      val_new := Roots.PolyEval(ADR(polynom), 5, tz);
      IF (ABS(val_new) < 64 * ABS(Roots.PolyEval(ADR(dderiv), 3, tz)) * Constants.Tolerance)
      THEN
        root[rootCount+1] := tz;
        rootCount := rootCount + 1;
      ELSIF (Roots.PolyEval(ADR(polynom), 5, tz_current) * val_new < 0)
      THEN
        root[rootCount+1] := Roots.ShrinkInterval(ADR(polynom), 5, tz_current, tz);
        rootCount := rootCount + 1;
      END_IF
    
      tz_current := tz;
    END_FOR
  
    val_max := Roots.PolyEval(ADR(polynom), 5, tz_max);
    IF Roots.PolyEval(ADR(polynom), 5, tz_current) * val_max < 0
    THEN
      root[rootCount+1] := Roots.ShrinkInterval(ADR(polynom), 5, tz_current, tz_max);
      rootCount := rootCount + 1;
    ELSIF ABS(val_max) < 8 * Constants.DoubleEpsilon
    THEN
      root[rootCount+1] := tz_max;
      rootCount := rootCount + 1;
    END_IF

    FOR i:=0 TO rootCount
    DO
      t := root[i];
      IF t < 0.0
      THEN
        CONTINUE;
      END_IF
    
      h1 := (a0_a0 + af_af)*0.5 + jMax*(2*a0*t + jMax*t*t - vd);
      IF h1 < 0
      THEN
        CONTINUE;
      END_IF
    
      IF ABS(jMax) < Constants.DoubleEpsilon
      THEN
        CONTINUE;
  		END_IF
    
      h1 := SQRT(h1)/ABS(jMax);
      orig := -pd - (2*a0_p3 + 4*af_p3 + 24*a0*jMax*t*(af + jMax*(h1 + t - tf)) + 6*a0_a0*(af + jMax*(2*t - tf)) + 6*(a0_a0 + af_af)*jMax*h1 + 12*af*jMax*(jMax*t*t - vd) + 12*jMax_jMax*(jMax*t*t*(h1 + t - tf) - tf*v0 - h1*vd))/(12*jMax_jMax);
      deriv_newton := -(a0 + jMax*t)*(3*(h1 + t) - 2*tf + (a0 + 2*af)/jMax);
    
      IF orig <> orig OR_ELSE deriv_newton <> deriv_newton OR_ELSE ABS(deriv_newton) < Constants.DoubleEpsilon 
      THEN
        CONTINUE;
      END_IF
    
      t := t - orig / deriv_newton;
  
      IF t > tf OR_ELSE t <> t (*isnan*)
      THEN
        CONTINUE;
      END_IF
  
      h1 := (a0_a0 + af_af)/(2*jMax_jMax) + (t*(2*a0 + jMax*t) - vd)/jMax;
      IF h1 >= 0
      THEN
        h1 := SQRT(h1);
    
        Profile.t[0] := t;
        Profile.t[1] := 0;
        Profile.t[2] := t + a0/jMax;
        Profile.t[3] := tf - 2*(t + h1) - (a0 + af)/jMax;
        Profile.t[4] := h1;
        Profile.t[5] := 0;
        Profile.t[6] := h1 + af/jMax;
    
        time_vel := Profile.CheckWithTiming(ProfileControlSigns.Uddu, ReachedLimits.vel, tf, jMax, vMax, vMin, aMax, aMin);
        IF time_vel
        THEN
          RETURN;
        END_IF
      END_IF
    END_FOR
  END_IF
  
  // Profile UDUD
  ph1 := af_af - 2*jMax*(2*af*tf + jMax*tf_tf - 3*vd);
  ph2 := af_p3 - 3*jMax_jMax*g1 + 3*af*jMax*vd;
  ph3 := 2*jMax*tf*g1 + 3*vd_vd;
  ph4 := af_p4 - 8*af_p3*jMax*tf + 12*jMax*(jMax*ph3 + af_af*vd + 2*af*jMax*(g1 - tf*vd));
  ph5 := af + jMax*tf;
  
  // Find root of 6th order polynom
  polynom[0] := 1.0;
  polynom[1] := (5*a0 - ph5)/jMax;
  polynom[2] := (39*a0_a0 - ph1 - 16*a0*ph5)/(4*jMax_jMax);
  polynom[3] := (55*a0_p3 - 33*a0_a0*ph5 - 6*a0*ph1 + 2*ph2)/(6*jMax_jMax*jMax);
  polynom[4] := (101*a0_p4 + ph4 - 76*a0_p3*ph5 - 30*a0_a0*ph1 + 16*a0*ph2)/(24*jMax_jMax*jMax_jMax);
  polynom[5] := (a0*(11*a0_p4 + ph4 - 10*a0_p3*ph5 - 6*a0_a0*ph1 + 4*a0*ph2))/(12*jMax_jMax*jMax_jMax*jMax);
  polynom[6] := (11*a0_p6 - af_p6 - 12*a0_p5*ph5 - 48*af_p3*jMax_jMax*g1 - 9*a0_p4*ph1 + 72*jMax_jMax*jMax*(jMax*g1*g1 - vd_vd*vd - 2*af*g1*vd) - 6*af_p4*jMax*vd - 36*af_af*jMax_jMax*vd_vd + 8*a0_p3*ph2 + 3*a0_a0*ph4)/(144*jMax_jMax*jMax_jMax*jMax_jMax);
  
  Roots.PolyMonicDeri(ADR(polynom), 6, out:=ADR(deriva));
  Roots.PolyMonicDeri(ADR(deriva), 5, out:=ADR(dderiv));
  Roots.SolveQuartMonic(ADR(dderiv[1]), 4, rootCount:=rootCount, roots:=root);
  
  tz_min := 0.0;
  tz_max := tf;
  dd_tz_current := tz_min;
  
  FOR i:=0 TO rootCount
  DO
    tz := root[i];
    IF tz >= tz_max
    THEN
      CONTINUE;
    END_IF
    
    orig := Roots.PolyEval(ADR(dderiv), 4, tz);
    IF (ABS(orig) > Constants.Tolerance)
    THEN
      Roots.PolyMonicDeri(ADR(dderiv), 4, out:=ADR(ddderiv));   
      res := Roots.PolyEval(ADR(ddderiv), 3, tz);
      IF ABS(res) > Constants.DoubleEpsilon
      THEN
        tz := tz - orig / res;
      END_IF
    END_IF  
  
    IF (Roots.PolyEval(ADR(deriva), 5, dd_tz_current) * Roots.PolyEval(ADR(deriva), 5, tz) < 0)
    THEN
      dd_tz_intervals[dd_tz_intervalCount+1, 0] := dd_tz_current;
      dd_tz_intervals[dd_tz_intervalCount+1, 1] := tz;
      dd_tz_intervalCount := dd_tz_intervalCount + 1;
    END_IF
  
    dd_tz_current := tz;
      
  END_FOR
  
  IF (Roots.PolyEval(ADR(deriva), 5, dd_tz_current) * Roots.PolyEval(ADR(deriva), 5, tz_max) < 0)
  THEN
    dd_tz_intervals[dd_tz_intervalCount+1, 0] := dd_tz_current; 
    dd_tz_intervals[dd_tz_intervalCount+1, 1] := tz_max;
    dd_tz_intervalCount := dd_tz_intervalCount + 1;
  END_IF
  
  rootCount := -1;
  tz_current := tz_min;
  FOR i:=0 TO dd_tz_intervalCount
  DO
    tz := Roots.ShrinkInterval(ADR(deriva), 5, dd_tz_intervals[i, 0], dd_tz_intervals[i, 1]);
    IF tz >= tz_max
    THEN
      CONTINUE;
    END_IF
    
    p_val := Roots.PolyEval(ADR(polynom), 6, tz);
    IF (ABS(p_val) < 64 * ABS(Roots.PolyEval(ADR(dderiv), 4, tz)) * Constants.Tolerance)
    THEN
      root[rootCount+1] := tz;
      rootCount := rootCount + 1;
    ELSIF (Roots.PolyEval(ADR(polynom), 6, tz_current) * p_val < 0)
    THEN
      root[rootCount+1] := Roots.ShrinkInterval(ADR(polynom), 6, tz_current, tz);
      rootCount := rootCount + 1;
    END_IF
    tz_current := tz;
  END_FOR
  
  IF (Roots.PolyEval(ADR(polynom), 6, tz_current) * Roots.PolyEval(ADR(polynom), 6, tz_max) < 0)
  THEN
    root[rootCount+1] := Roots.ShrinkInterval(ADR(polynom), 6, tz_current, tz_max);
    rootCount := rootCount + 1;
  END_IF
  
  
  FOR i:=0 TO rootCount
  DO
    t := root[i];
    
    // Double Newton step (regarding pd)
    h1 := (af_af - a0_a0)/(2*jMax_jMax) - ((2*a0 + jMax*t)*t - vd)/jMax;
    IF h1 < 0
    THEN
      CONTINUE;
    END_IF
    
    h1 := SQRT(h1);
    orig := -pd + (af_p3 - a0_p3 + 3*a0_a0*jMax*(tf - 2*t))/(6*jMax_jMax) + (2*a0 + jMax*t)*t*(tf - t) + (jMax*h1 - af)*h1*h1 + tf*v0;
    deriv_newton := (a0 + jMax*t)*(2*(af + jMax*tf) - 3*jMax*(h1 + t) - a0)/jMax;
  
    IF ABS(deriv_newton) <= Constants.DoubleEpsilon
    THEN
      CONTINUE;
    END_IF
    
    t := t - orig / deriv_newton;
    h1 := (af_af - a0_a0)*0.5 - jMax*((2*a0 + jMax*t)*t - vd);
    IF h1 < 0
    THEN
      CONTINUE;
    END_IF
    h1 := SQRT(h1)/ABS(jMax);  
    orig := -pd + (af_p3 - a0_p3 + 3*a0_a0*jMax*(tf - 2*t))/(6*jMax_jMax) + (2*a0 + jMax*t)*t*(tf - t) + (jMax*h1 - af)*h1*h1 + tf*v0;
    IF (ABS(orig) > 1E-9)
    THEN
      deriv_newton := (a0 + jMax*t)*(2*(af + jMax*tf) - 3*jMax*(h1 + t) - a0)/jMax;
      
      IF ABS(deriv_newton) <= Constants.DoubleEpsilon
      THEN
        CONTINUE;
      END_IF
      
      t := t - orig / deriv_newton;           
    END_IF
  
    h1 := (af_af - a0_a0)*0.5 - jMax*((2*a0 + jMax*t)*t - vd);
    IF h1 < 0
    THEN
      CONTINUE;
    END_IF
    h1 := SQRT(h1)/ABS(jMax);
    Profile.t[0] := t;
    Profile.t[1] := 0;
    Profile.t[2] := t + a0/jMax;
    Profile.t[3] := tf - 2*(t + h1) + ad/jMax;
    Profile.t[4] := h1;
    Profile.t[5] := 0;
    Profile.t[6] := h1 - af/jMax;
  
    time_vel := Profile.CheckWithTiming(ProfileControlSigns.Udud, ReachedLimits.Vel, tf, jMax, vMax, vMin, aMax, aMin);
    IF time_vel
    THEN
      RETURN;
    END_IF
  END_FOR
END_IF
END_METHOD

END_FUNCTION_BLOCK

// ---- Struckig/Math/Power2.TcPOU
// Struckig
// Copyright (C) 2022 Stefan Besler

// This program is free software: you can redistribute it and/or modify
// it under the terms of the GNU General Public License as published by
// the Free Software Foundation, either version 3 of the License, or
// (at your option) any later version.

// This program is distributed in the hope that it will be useful,
// but WITHOUT ANY WARRANTY; without even the implied warranty of
// MERCHANTABILITY or FITNESS FOR A PARTICULAR PURPOSE.  See the
// GNU General Public License for more details.
//
// You should have received a copy of the GNU General Public License
// along with THIS PROGRAM.  IF NOT, see <http://www.gnu.org/licenses/>.
/// Internal square helper.
/// Returns `v * v`.
FUNCTION INTERNAL Power2 : LREAL
VAR_INPUT
  v : LREAL; //< Input value.
END_VAR

Power2 := v*v;

END_FUNCTION

// ---- Struckig/Velocity/VelocityThirdOrderStep1.TcPOU
// Struckig
// Copyright (C) 2022 Stefan Besler

// This program is free software: you can redistribute it and/or modify
// it under the terms of the GNU General Public License as published by
// the Free Software Foundation, either version 3 of the License, or
// (at your option) any later version.

// This program is distributed in the hope that it will be useful,
// but WITHOUT ANY WARRANTY; without even the implied warranty of
// MERCHANTABILITY or FITNESS FOR A PARTICULAR PURPOSE.  See the
// GNU General Public License for more details.
//
// You should have received a copy of the GNU General Public License
// along with THIS PROGRAM.  IF NOT, see <http://www.gnu.org/licenses/>.
/// Mathematical equations for Step 1 in third-order velocity interface: Extremal profiles
FUNCTION_BLOCK INTERNAL VelocityThirdOrderStep1 
VAR
  a0, af : LREAL;
  aMax, aMin, jMax : LREAL;
  vd : LREAL;
  
  ValidProfiles : ARRAY[0..2] OF ProfileDesc; // Max 3 valid profiles
  ValidProfileCount : INT := -1;  
END_VAR

METHOD AddInterval
VAR_INPUT
  interval : REFERENCE TO BlockInterval;
  Left : REFERENCE TO ProfileDesc;
  Right : REFERENCE TO ProfileDesc;
END_VAR
VAR_INST
  left_duration,right_duration : LREAL;   
END_VAR
left_duration := Left.t_sum[6] + Left.Brake.Duration + Left.Accel.Duration; 
right_duration := Right.t_sum[6] + Right.Brake.Duration + Right.Accel.Duration; 
IF (left_duration < right_duration)
THEN
  interval.Left := left_duration;
  interval.Right := right_duration;
  interval.Profile := Right;
  interval.IsUsed := TRUE;
ELSE
  interval.Left := right_duration;
  interval.Right := left_duration;
  interval.Profile := Left;
  interval.IsUsed := TRUE;
END_IF
END_METHOD

METHOD AddProfile
VAR_IN_OUT CONSTANT
  Profile : ProfileDesc;
END_VAR
ValidProfileCount := ValidProfileCount + 1;
ValidProfiles[ValidProfileCount] := Profile;
ValidProfiles[ValidProfileCount].pf := Profile.p[7];
END_METHOD

METHOD CalculateBlock : BOOL
VAR_INPUT
  block : REFERENCE TO Block;
END_VAR
VAR
  i, j : INT;
  Tmin : LREAL;
  idx_min : INT;
  idx_else_1, idx_else_2, idx_else_3, idx_else_4 : INT;
END_VAR
IF (ValidProfileCount = 0) OR_ELSE (ValidProfileCount = 1 AND_THEN ABS(ValidProfiles[0].t_sum[6] - ValidProfiles[1].t_sum[6]) < 8*Constants.Epsilon)
THEN
  block.Pmin := ValidProfiles[0];
  block.Tmin := block.Pmin.t_sum[6] + block.Pmin.Brake.Duration + block.Pmin.Accel.Duration;  
  CalculateBlock := TRUE;
  RETURN;
// Only happens due to numerical issues
ELSIF (ValidProfileCount = 3) 
THEN
  // Find "identical" profiles
  IF (ABS(ValidProfiles[0].t_sum[6] - ValidProfiles[1].t_sum[6]) < 16*Constants.Epsilon OR_ELSE ValidProfiles[0].Direction <> ValidProfiles[1].Direction)
  THEN
    RemoveProfile(1);
  ELSIF (ABS(ValidProfiles[1].t_sum[6] - ValidProfiles[2].t_sum[6]) < 16*Constants.Epsilon  OR_ELSE ValidProfiles[2].Direction <> ValidProfiles[2].Direction)
  THEN
    RemoveProfile(2);
  ELSIF (ABS(ValidProfiles[0].t_sum[6] - ValidProfiles[2].t_sum[6]) < 256*Constants.Epsilon OR_ELSE ValidProfiles[0].Direction <> ValidProfiles[2].Direction)
  THEN
    RemoveProfile(2);
  ELSE
    RETURN;
  END_IF

ELSIF ((ValidProfileCount+1) MOD 2 = 0)
THEN
  RETURN;
END_IF

// Find index of fastest Profile
Tmin := Constants.Infinity;
FOR i:=0 TO ValidProfileCount
DO
  FOR j:=0 TO ValidProfileCount
  DO
    IF ValidProfiles[i].t_sum[6] + ValidProfiles[i].Brake.Duration < ValidProfiles[j].t_sum[6] + ValidProfiles[j].Brake.Duration AND_THEN
       ValidProfiles[i].t_sum[6] + ValidProfiles[i].Brake.Duration < Tmin
    THEN
      Tmin := ValidProfiles[i].t_sum[6] + ValidProfiles[i].Brake.Duration + ValidProfiles[i].Accel.Duration;
      idx_min := i;
		END_IF
  END_FOR
END_FOR

block.Pmin := ValidProfiles[idx_min];
block.Tmin := block.Pmin.t_sum[6] + block.Pmin.Brake.Duration + block.Pmin.Accel.Duration;  

IF (ValidProfileCount = 2)
THEN
  idx_else_1 := (idx_min + 1) MOD 3;
  idx_else_2 := (idx_min + 2) MOD 3;
  
  AddInterval(block.A, ValidProfiles[idx_else_1], ValidProfiles[idx_else_2]);
  CalculateBlock := TRUE;
  RETURN;

 ELSIF (ValidProfileCount = 4)
 THEN
  idx_else_1 := (idx_min + 1) MOD 5;
  idx_else_2 := (idx_min + 2) MOD 5;
  idx_else_3 := (idx_min + 3) MOD 5;
  idx_else_4 := (idx_min + 4) MOD 5;
  
  IF (ValidProfiles[idx_else_1].Direction = ValidProfiles[idx_else_2].Direction)
  THEN
    AddInterval(block.A, ValidProfiles[idx_else_1], ValidProfiles[idx_else_2]);
    AddInterval(block.B, ValidProfiles[idx_else_3], ValidProfiles[idx_else_4]);
  ELSE 
    AddInterval(block.A, ValidProfiles[idx_else_1], ValidProfiles[idx_else_4]);
    AddInterval(block.B, ValidProfiles[idx_else_2], ValidProfiles[idx_else_3]);
  END_IF
  
  CalculateBlock := TRUE;
  RETURN;
END_IF
END_METHOD

METHOD Get : BOOL
VAR_INPUT
  input : ProfileDesc;
END_VAR
VAR_IN_OUT
  block : Block; 
END_VAR
VAR
  aMax, aMin, jMax : LREAL;
END_VAR
ValidProfileCount := -1;

// Zero-limits special case
IF THIS^.jMax = 0.0
THEN
  block.Pmin.SetBoundary(input);
  
  IF time_all_single_step(block.Pmin, THIS^.aMax, THIS^.aMin, THIS^.jMax)
  THEN
    block.Tmin := block.Pmin.t_sum[6] + block.Pmin.Brake.Duration + block.Pmin.Accel.Duration;
    AddInterval(block.A, block.Pmin, block.Pmin);
    IF ABS(a0) > Constants.DoubleEpsilon
    THEN
	  block.A.Left := block.Tmin;
      block.A.Right := Constants.Infinity;
    END_IF
    
    Get := TRUE;
    RETURN; 
	END_IF
  
  RETURN;  
END_IF

validProfiles[0].SetBoundary(input);

IF ABS(af) < Constants.DoubleEpsilon
THEN
  // There is no blocked interval when af==0, so return after first found profile
  aMax := SEL((vd >= 0), THIS^.aMin, THIS^.aMax);
  aMin := SEL((vd >= 0), THIS^.aMax, THIS^.aMin);
  jMax := SEL((vd >= 0), -THIS^.jMax, THIS^.jMax);
  
  time_none(input, aMax, aMin, jMax, TRUE);
  IF ValidProfileCount >= 0
  THEN 
    Get := CalculateBlock(block);
    RETURN;
	END_IF
  
  time_acc0(input, aMax, aMin, jMax, TRUE);
  IF ValidProfileCount >= 0
  THEN 
    Get := CalculateBlock(block);
    RETURN;
	END_IF
  
  time_none(input, aMin, aMax, -jMax, TRUE);
  IF ValidProfileCount >= 0
  THEN 
    Get := CalculateBlock(block);
    RETURN;
	END_IF
  
  time_acc0(input, aMin, aMax, -jMax, TRUE);
ELSE
  time_none(input, THIS^.aMax, THIS^.aMin, THIS^.jMax, FALSE);
  time_none(input, THIS^.aMin, THIS^.aMax, -THIS^.jMax, FALSE);
  time_acc0(input, THIS^.aMax, THIS^.aMin, THIS^.jMax, FALSE);
  time_acc0(input, THIS^.aMin, THIS^.aMax, -THIS^.jMax, FALSE);
END_IF

Get := CalculateBlock(block);
END_METHOD

METHOD PRIVATE RemoveProfile : BOOL
VAR_INPUT
  index : INT;
END_VAR
VAR
  i : INT;
END_VAR
// todo, this is pretty slow in twincat
FOR i:=index TO ValidProfileCount-2
DO
  ValidProfiles[i] := ValidProfiles[i + 1];
END_FOR

ValidProfileCount := ValidProfileCount - 1;
END_METHOD

METHOD Set
VAR_INPUT
  v0, a0 : LREAL; 
  vf, af : LREAL; 
  aMax, aMin : LREAL; 
  jMax : LREAL;   
END_VAR
THIS^.a0 := a0;
THIS^.vd := vf - v0;
THIS^.af := af;;
THIS^.aMax := aMax;
THIS^.aMin := aMin;
THIS^.jMax := jMax;
END_METHOD

METHOD PRIVATE time_acc0
VAR_IN_OUT
  profile : ProfileDesc;
END_VAR
VAR_INPUT
  aMax, aMin, jMax : LREAL;
  return_after_found : BOOL;  
END_VAR
// UD
profile.t[0] := (-a0 + aMax)/jMax;
profile.t[1] := (a0*a0 + af*af - 2*aMax*aMax + 2*jMax*vd)/(2*aMax*jMax);
profile.t[2] := (-af + aMax)/jMax;
profile.t[3] := 0;
profile.t[4] := 0;
profile.t[5] := 0;
profile.t[6] := 0;

IF (Profile.CheckForVelocity(ProfileControlSigns.Uddu, ReachedLimits.Acc0, jMax, aMax, aMin))
THEN
  AddProfile(profile);
  IF return_after_found
  THEN
    RETURN;
	END_IF
END_IF
END_METHOD

METHOD PRIVATE time_all_single_step : BOOL
VAR_IN_OUT
  profile : ProfileDesc;
END_VAR
VAR_INPUT
  aMax, aMin, jMax : LREAL;
END_VAR
IF ABS(af - a0) > Constants.DoubleEpsilon
THEN 
  RETURN;
END_IF
    
profile.t[0] := 0;
profile.t[1] := 0;
profile.t[2] := 0;
profile.t[3] := 0;
profile.t[4] := 0;
profile.t[5] := 0;
profile.t[6] := 0;

IF ABS(a0) > Constants.DoubleEpsilon
THEN

  IF ABS(a0) > Constants.DoubleEpsilon
  THEN
    profile.t[3] := vd / a0;
    IF profile.CheckForVelocity(ProfileControlSigns.uddu, ReachedLimits.None, 0.0, aMax, aMin)
    THEN
      time_all_single_step := TRUE;
      RETURN;
    END_IF
	END_IF

 ELSE IF ABS(vd) < Constants.DoubleEpsilon
 THEN
    IF profile.CheckForVelocity(ProfileControlSigns.uddu, ReachedLimits.None, 0.0, aMax, aMin)
    THEN 
      time_all_single_step := TRUE;
      RETURN;
  END_IF
 END_IF
END_IF
END_METHOD

METHOD PRIVATE time_none
VAR_IN_OUT
  profile : ProfileDesc;
END_VAR
VAR_INPUT
  aMax, aMin, jMax : LREAL;
  return_after_found : BOOL;    
END_VAR
VAR
  h1 : LREAL;
END_VAR
h1 := (a0*a0 + af*af)/2 + jMax*vd;
IF h1>=0
THEN
  h1 := SQRT(h1);
  
  // Solution 1
  profile.t[0] := -(a0 + h1)/jMax;
  profile.t[1] := 0;
  profile.t[2] := -(af + h1)/jMax;
  profile.t[3] := 0;
  profile.t[4] := 0;
  profile.t[5] := 0;
  profile.t[6] := 0;  
  
  IF (profile.CheckForVelocity(ProfileControlSigns.uddu, ReachedLimits.None, jMax, aMax, aMin))
  THEN
    AddProfile(profile);
    IF return_after_found
    THEN
      RETURN;
    END_IF
  END_IF

  // Solution 2
  profile.t[0] := (-a0 + h1)/jMax;
  profile.t[1] := 0;
  profile.t[2] := (-af + h1)/jMax;
  profile.t[3] := 0;
  profile.t[4] := 0;
  profile.t[5] := 0;
  profile.t[6] := 0;    
  
  IF (profile.CheckForVelocity(ProfileControlSigns.uddu, ReachedLimits.None, jMax, aMax, aMin)) THEN
    AddProfile(profile);  
  END_IF
END_IF
END_METHOD

END_FUNCTION_BLOCK

// ---- Struckig/Velocity/VelocityThirdOrderStep2.TcPOU
// Struckig
// Copyright (C) 2022 Stefan Besler

// This program is free software: you can redistribute it and/or modify
// it under the terms of the GNU General Public License as published by
// the Free Software Foundation, either version 3 of the License, or
// (at your option) any later version.

// This program is distributed in the hope that it will be useful,
// but WITHOUT ANY WARRANTY; without even the implied warranty of
// MERCHANTABILITY or FITNESS FOR A PARTICULAR PURPOSE.  See the
// GNU General Public License for more details.
//
// You should have received a copy of the GNU General Public License
// along with THIS PROGRAM.  IF NOT, see <http://www.gnu.org/licenses/>.
/// Mathematical equations for Step 2 in third-order velocity interface: Time synchronization
FUNCTION_BLOCK INTERNAL VelocityThirdOrderStep2 
VAR
  tf, a0, af, vd, ad : LREAL;
  aMax, aMin, jMax : LREAL;
END_VAR

METHOD CheckAll : BOOL
VAR_IN_OUT
  Profile : ProfileDesc;
END_VAR
VAR_INPUT
  aMax, aMin, jMax : LREAL;
END_VAR
CheckAll := time_acc0(Profile, aMax, aMin, jMax) OR_ELSE time_none(Profile, aMax, aMin, jMax);
END_METHOD

METHOD Get : BOOL
VAR_IN_OUT
  Profile : ProfileDesc;
END_VAR
// Test all cases to get ones that match
// However we should guess which one is correct and try them first...
IF (vd > 0) THEN
  Get := CheckAll(Profile, aMax, aMin, jMax) OR_ELSE CheckAll(Profile, aMin, aMax, -jMax);
ELSE
  Get := CheckAll(Profile, aMin, aMax, -jMax) OR_ELSE CheckAll(Profile, aMax, aMin, jMax);
END_IF
END_METHOD

METHOD Set
VAR_INPUT
  tf : LREAL;
  v0, a0 : LREAL;
  vf, af : LREAL;
  aMax, aMin : LREAL;
  jMax : LREAL; 
END_VAR
THIS^.a0 := a0;
THIS^.tf := tf;
THIS^.af := af;
THIS^.aMax := aMax;
THIS^.aMin := aMin;
THIS^.jMax := jMax;
THIS^.vd := vf - v0;
THIS^.ad := af - a0;
END_METHOD

METHOD PRIVATE time_acc0 : BOOL
VAR_IN_OUT
  profile : ProfileDesc;
END_VAR
VAR_INPUT
  aMax, aMin, jMax : LREAL;
END_VAR
VAR
  h1 : LREAL;
END_VAR
// UD Solution 1/2
h1 := (-a0*a0 - af*af + 2*a0*af + 2*jMax*((a0 + af)*tf - 2*(vd)))/(jMax*jMax) + tf*tf;
IF h1 >= 0
THEN
  h1 := SQRT(h1);
  
  profile.t[0] := ad/(2*jMax) + (tf - h1)/2;
  profile.t[1] := h1;
  profile.t[2] := tf - (profile.t[0] + h1);
  profile.t[3] := 0;
  profile.t[4] := 0;
  profile.t[5] := 0;
  profile.t[6] := 0;
  
  IF (profile.CheckForVelocity(ProfileControlSigns.uddu, ReachedLimits.Acc0, jMax, aMax, aMin)) THEN
    profile.pf := profile.p[7];
    time_acc0 := TRUE;
    RETURN;
  END_IF
END_IF

// UU Solution
h1 := (jMax*tf - ad);

IF ABS(h1) > Constants.Epsilon AND_THEN ABS(2*jMax*h1) > Constants.Epsilon
THEN
  profile.t[0] := -ad*ad/(2*jMax*h1) + (vd - a0*tf)/h1;
  profile.t[1] := -ad/jMax + tf;
  profile.t[2] := 0;
  profile.t[3] := 0;
  profile.t[4] := 0;
  profile.t[5] := 0;
  profile.t[6] := tf - (profile.t[0] + profile.t[1]);

  IF (profile.CheckForVelocity(ProfileControlSigns.Uddu, ReachedLimits.Acc0, jMax, aMax, aMin))
  THEN
    profile.pf := profile.p[7];
    time_acc0 := TRUE;
    RETURN;
  END_IF
END_IF

// UU Solution - 2 step
profile.t[0] := 0;
profile.t[1] := -ad/jMax + tf;
profile.t[2] := 0;
profile.t[3] := 0;
profile.t[4] := 0;
profile.t[5] := 0;
profile.t[6] := ad/jMax;

IF (profile.CheckForVelocity(ProfileControlSigns.Uddu, ReachedLimits.Acc0, jMax, aMax, aMin))
THEN
  profile.pf := profile.p[7];
  time_acc0 := TRUE;
  RETURN;
END_IF
END_METHOD

METHOD PRIVATE time_none : BOOL
VAR_IN_OUT
  profile : ProfileDesc;
END_VAR
VAR_INPUT
  aMax, aMin, jMax : LREAL;
END_VAR
VAR
  h1, jf : LREAL;
END_VAR
IF (ABS(a0) < Constants.DoubleEpsilon AND_THEN ABS(af) < Constants.DoubleEpsilon AND_THEN ABS(vd) < Constants.DoubleEpsilon) THEN
  profile.t[0] := 0;
  profile.t[1] := tf;
  profile.t[2] := 0;
  profile.t[3] := 0;
  profile.t[4] := 0;
  profile.t[5] := 0;
  profile.t[6] := 0;
  
  IF (profile.CheckForVelocity(ProfileControlSigns.uddu, ReachedLimits.None, jMax, aMax, aMin)) THEN
    profile.pf := profile.p[7];
    time_none := TRUE;
    RETURN;
  END_IF
END_IF
    
// UD Solution 1/2
h1 := 2*(af*tf - vd);
IF ABS(af - a0) > Constants.DoubleEpsilon AND_THEN ABS(h1) > Constants.Epsilon
THEN
  profile.t[0] := h1/(af - a0);
  profile.t[1] := tf - profile.t[0];
  profile.t[2] := 0;
  profile.t[3] := 0;
  profile.t[4] := 0;
  profile.t[5] := 0;
  profile.t[6] := 0;
  
  jf := Power2(a0 - af)/h1;
  IF (ABS(jf) < ABS(jMax) + 1E-12 AND_THEN profile.CheckForVelocity(ProfileControlSigns.uddu, ReachedLimits.None, jf, aMax, aMin))
  THEN
    profile.pf := profile.p[7];
    time_none := TRUE;
  END_IF
END_IF
END_METHOD

END_FUNCTION_BLOCK

// ---- Struckig/Position/PositionSecondOrderStep1.TcPOU
// Struckig
// Copyright (C) 2022 Stefan Besler

// This program is free software: you can redistribute it and/or modify
// it under the terms of the GNU General Public License as published by
// the Free Software Foundation, either version 3 of the License, or
// (at your option) any later version.

// This program is distributed in the hope that it will be useful,
// but WITHOUT ANY WARRANTY; without even the implied warranty of
// MERCHANTABILITY or FITNESS FOR A PARTICULAR PURPOSE.  See the
// GNU General Public License for more details.
//
// You should have received a copy of the GNU General Public License
// along with THIS PROGRAM.  IF NOT, see <http://www.gnu.org/licenses/>.
/// Mathematical equations for Step 1 in third-order position interface: Extremal profiles
FUNCTION_BLOCK INTERNAL PositionSecondOrderStep1
VAR
  v0 : LREAL;
  vf : LREAL;
  _vMax, _vMin, _aMax, _aMin : LREAL;

  // Pre-calculated expressions
  pd : LREAL;
  h1 : LREAL;
  
  validProfiles : ARRAY[0..5] OF ProfileDesc; // Max 5 valid profiles + 1 spare for numerical issues
  validProfileCounter : INT := -1;
  
  left_duration, right_duration : LREAL;    
END_VAR

METHOD AddInterval
VAR_IN_OUT
  interval : BlockInterval;
  Left : ProfileDesc;
  Right : ProfileDesc;
END_VAR
left_duration := Left.t_sum[6] + Left.Brake.Duration + Left.Accel.Duration;
right_duration := Right.t_sum[6] + Right.Brake.Duration + Right.Accel.Duration;
IF (left_duration < right_duration)
THEN
  interval.Left := left_duration;
  interval.Right := right_duration;
  interval.Profile := Right;
  interval.IsUsed := TRUE;
ELSE
  interval.Left := right_duration;
  interval.Right := left_duration;
  interval.Profile := Left;
  interval.IsUsed := TRUE;  
END_IF
END_METHOD

METHOD AddProfile
VAR_IN_OUT CONSTANT
  Profile : ProfileDesc;
END_VAR
validProfileCounter := validProfileCounter + 1;
validProfiles[validProfileCounter] := Profile;
END_METHOD

METHOD CalculateBlock : BOOL
VAR_IN_OUT
  block : Block;
END_VAR
VAR
  i, j : INT;
  Tmin : LREAL;
  idx_min : INT;
  idx_else_1, idx_else_2, idx_else_3, idx_else_4 : INT;
END_VAR
block.A.IsUsed := FALSE;
block.B.IsUsed := FALSE;

IF validProfileCounter = 0
THEN
  block.Pmin := validProfiles[0];
  block.Tmin := block.Pmin.t_sum[6] + block.Pmin.Brake.Duration + block.Pmin.Accel.Duration; 
  CalculateBlock := TRUE;

ELSIF validProfileCounter = 1 
THEN

  IF ABS(validProfiles[0].t_sum[6] - validProfiles[1].t_sum[6]) < 8*Constants.Epsilon
  THEN
    block.Pmin := validProfiles[0];
    block.Tmin := block.Pmin.t_sum[6] + block.Pmin.Brake.Duration + block.Pmin.Accel.Duration;  
    CalculateBlock := TRUE;
    RETURN;
	END_IF
  
  IF ParameterList.NumericalRobust
  THEN
    idx_min := SEL(validProfiles[0].t_sum[6] < validProfiles[1].t_sum[6], 1, 0);
    idx_else_1 := (idx_min + 1) MOD 2;

    block.Pmin := validProfiles[idx_min];
    block.Tmin := block.Pmin.t_sum[6] + block.Pmin.Brake.Duration + block.Pmin.Accel.Duration; 
    AddInterval(block.A, validProfiles[idx_min], validProfiles[idx_else_1]);
    CalculateBlock := TRUE;
    RETURN; 
	END_IF

// Only happens due to numerical issues
ELSIF (validProfileCounter = 3) 
THEN
  // Find "identical" profiles
  IF (ABS(validProfiles[0].t_sum[6] - validProfiles[1].t_sum[6]) < 32*Constants.Epsilon AND_THEN validProfiles[0].Direction <> validProfiles[1].Direction)
  THEN
    RemoveProfile(1);
  ELSIF (ABS(validProfiles[2].t_sum[6] - validProfiles[3].t_sum[6]) < 256*Constants.Epsilon  AND_THEN validProfiles[2].Direction <> validProfiles[3].Direction)
  THEN
    RemoveProfile(3);
  ELSIF (ABS(validProfiles[0].t_sum[6] - validProfiles[3].t_sum[6]) < 256*Constants.Epsilon AND_THEN validProfiles[0].Direction <> validProfiles[3].Direction)
  THEN
    RemoveProfile(3);
  ELSE
    RETURN;
  END_IF

ELSIF ((validProfileCounter+1) MOD 2 = 0)
THEN
  RETURN;
END_IF

// Find index of fastest Profile
Tmin := Constants.Infinity;
FOR i:=0 TO validProfileCounter
DO
  FOR j:=0 TO validProfileCounter
  DO
    IF validProfiles[i].t_sum[6] + validProfiles[i].Brake.Duration < validProfiles[j].t_sum[6] + validProfiles[j].Brake.Duration AND_THEN
       validProfiles[i].t_sum[6] + validProfiles[i].Brake.Duration < Tmin
    THEN
      Tmin := validProfiles[i].t_sum[6] + validProfiles[i].Brake.Duration + validProfiles[i].Accel.Duration;
      idx_min := i;
		END_IF
  END_FOR
END_FOR

block.Pmin := validProfiles[idx_min];
block.Tmin := block.Pmin.t_sum[6] + block.Pmin.Brake.Duration + block.Pmin.Accel.Duration;
IF (validProfileCounter = 2)
THEN
  idx_else_1 := (idx_min + 1) MOD 3;
  idx_else_2 := (idx_min + 2) MOD 3;
  
  AddInterval(block.A, validProfiles[idx_else_1], validProfiles[idx_else_2]);
  CalculateBlock := TRUE;
  RETURN;

 ELSIF (validProfileCounter = 4)
 THEN
  idx_else_1 := (idx_min + 1) MOD 5;
  idx_else_2 := (idx_min + 2) MOD 5;
  idx_else_3 := (idx_min + 3) MOD 5;
  idx_else_4 := (idx_min + 4) MOD 5;
  
  IF (validProfiles[idx_else_1].Direction = validProfiles[idx_else_2].Direction)
  THEN
    AddInterval(block.A, validProfiles[idx_else_1], validProfiles[idx_else_2]);
    AddInterval(block.B, validProfiles[idx_else_3], validProfiles[idx_else_4]);
  ELSE 
    AddInterval(block.A, validProfiles[idx_else_1], validProfiles[idx_else_4]);
    AddInterval(block.B, validProfiles[idx_else_2], validProfiles[idx_else_3]);
  END_IF
  
  CalculateBlock := TRUE;
END_IF
END_METHOD

METHOD Get : BOOL
VAR_INPUT
  input : REFERENCE TO ProfileDesc;
  block : REFERENCE TO Block; 
END_VAR
VAR_INST
  vMax, vMin, aMax, aMin, jMax : LREAL;
  profile : REFERENCE TO ProfileDesc;
END_VAR
validProfileCounter := -1;

// Zero-limits special case
IF _vMax = 0.0 AND_THEN _vMin = 0.0
THEN
  block.Pmin.SetBoundary(input);

  IF time_all_single_step(block.Pmin, _vMax, _vMin, _aMax, _aMin) 
  THEN
    block.Tmin := block.Pmin.t_sum[6] + block.Pmin.Brake.Duration + block.Pmin.Accel.Duration;
    AddInterval(block.A, block.Pmin, block.Pmin);
    
    IF ABS(v0) > Constants.DoubleEpsilon 
    THEN
	    block.A.Left := block.Tmin;
      block.A.Right := Constants.Infinity;
    END_IF
    
    Get := TRUE;
    RETURN; 
  END_IF
  
  RETURN;
END_IF

validProfiles[0].SetBoundary(input);

IF ABS(vf) < Constants.DoubleEpsilon
THEN
  // There is no blocked interval when vf==0, so return after first found profile
  vMax := SEL(pd >= 0, _vMin, _vMax);
  vMin := SEL(pd >= 0, _vMax, _vMin);
  aMax := SEL(pd >= 0, _aMin, _aMax);
  aMin := SEL(pd >= 0, _aMax, _aMin);
  
  time_none(input, vMax, vMin, aMax, aMin, TRUE);
  IF (validProfileCounter >= 0) THEN
    Get := CalculateBlock(block);
    RETURN;
  END_IF
  
  time_acc0(input, vMax, vMin, aMax, aMin, TRUE);
  IF (validProfileCounter >= 0) THEN
    Get := CalculateBlock(block);
    RETURN;
  END_IF
  
  time_none(input, vMin, vMax, aMin, aMax, TRUE);
  IF (validProfileCounter >= 0) THEN
    Get := CalculateBlock(block);
    RETURN;
  END_IF
  
  time_acc0(input, vMin, vMax, aMin, aMax, TRUE);
  IF (validProfileCounter >= 0) THEN
    Get := CalculateBlock(block);
    RETURN;
  END_IF 
ELSE
  time_none(input, _vMax, _vMin, _aMax, _aMin, FALSE);
  time_none(input, _vMin, _vMax, _aMin, _aMax, FALSE);
  time_acc0(input, _vMax, _vMin, _aMax, _aMin, FALSE);
  time_acc0(input, _vMin, _vMax, _aMin, _aMax, FALSE);
  
  IF (validProfileCounter >= 0) THEN
    Get := CalculateBlock(block);
    RETURN;
  END_IF   
END_IF
END_METHOD

METHOD PRIVATE RemoveProfile : BOOL
VAR_INPUT
  index : INT;
END_VAR
VAR
  i : INT;
END_VAR
// todo, this is pretty slow in twincat
FOR i:=index TO validProfileCounter-2
DO
  validProfiles[i] := validProfiles[i + 1];
END_FOR

validProfileCounter := validProfileCounter - 1;
END_METHOD

METHOD Set
VAR_INPUT
  p0, v0 : LREAL;
  pf, vf : LREAL;
  vMax, vMin : LREAL;
  aMax, aMin : LREAL;
END_VAR
THIS^.v0 := v0;
THIS^.vf := vf;
THIS^._vMax := vMax;
THIS^._vMin := vMin;
THIS^._aMax := aMax;
THIS^._aMin := aMin;

pd := pf - p0;
END_METHOD

METHOD PRIVATE time_acc0
VAR_INPUT
  profile : REFERENCE TO ProfileDesc;
  vMax, vMin, aMax, aMin : LREAL;
  return_after_found : BOOL;  
END_VAR
profile.t[0] := (-v0 + vMax)/aMax;
profile.t[1] :=(aMin*v0*v0 - aMax*vf*vf)/(2*aMax*aMin*vMax) + vMax*(aMax - aMin)/(2*aMax*aMin) + pd/vMax;
profile.t[2] := (vf - vMax)/aMin;
profile.t[3] := 0;
profile.t[4] := 0;
profile.t[5] := 0;
profile.t[6] := 0;

IF profile.CheckForSecondOrder(ProfileControlSigns.Uddu, ReachedLimits.Acc0, aMax, aMin, vMax, vMin)
THEN
  AddProfile(profile);
END_IF
END_METHOD

METHOD PRIVATE time_all_single_step : BOOL
VAR_INPUT
  profile : REFERENCE TO ProfileDesc;
  vMax, vMin, aMax, aMin : LREAL;
END_VAR
IF ABS(vf - v0) > Constants.DoubleEpsilon
THEN
  RETURN;
END_IF

profile.t[0] := 0;
profile.t[1] := 0;
profile.t[2] := 0;
profile.t[3] := 0;
profile.t[4] := 0;
profile.t[5] := 0;
profile.t[6] := 0;

IF ABS(v0) > Constants.DoubleEpsilon
THEN
  profile.t[3] := pd / v0;
  IF (profile.CheckForSecondOrder(ProfileControlSigns.Uddu, ReachedLimits.None, 0.0, 0.0, vMax, vMin))
  THEN
    time_all_single_step := TRUE;
  END_IF
ELSIF ABS(pd) < Constants.DoubleEpsilon
THEN
  IF (profile.CheckForSecondOrder(ProfileControlSigns.Uddu, ReachedLimits.None, 0.0, 0.0, vMax, vMin))
  THEN
    time_all_single_step := TRUE;
  END_IF
END_IF
END_METHOD

/// Only for numerical issues, always return_after_found
METHOD PRIVATE time_none
VAR_INPUT
  profile : REFERENCE TO ProfileDesc;
  vMax, vMin, aMax, aMin : LREAL;
  return_after_found : BOOL;
END_VAR
h1 := (aMax*vf*vf - aMin*v0*v0 - 2*aMax*aMin*pd)/(aMax - aMin);
IF h1 >= 0.0
THEN
  h1 := SQRT(h1);
  
  // Solution 1
  profile.t[0] := -(v0 + h1)/aMax;
  profile.t[1] := 0;
  profile.t[2] := (vf + h1)/aMin;
  profile.t[3] := 0;
  profile.t[4] := 0;
  profile.t[5] := 0;
  profile.t[6] := 0;  
  IF profile.CheckForSecondOrder(ProfileControlSigns.Uddu, ReachedLimits.None, aMax, aMin, vMax, vMin)
  THEN
    AddProfile(profile);
    IF return_after_found
    THEN
      RETURN;
    END_IF
  END_IF

  
  // Solution 2
  profile.t[0] := (-v0 + h1)/aMax;
  profile.t[1] := 0;
  profile.t[2] := (vf - h1)/aMin;
  profile.t[3] := 0;
  profile.t[4] := 0;
  profile.t[5] := 0;
  profile.t[6] := 0;  
  IF profile.CheckForSecondOrder(ProfileControlSigns.Uddu, ReachedLimits.None, aMax, aMin, vMax, vMin)
  THEN
    AddProfile(profile);
    IF return_after_found
    THEN
      RETURN;
    END_IF
  END_IF
END_IF
END_METHOD

END_FUNCTION_BLOCK

// ---- Struckig/Position/PositionSecondOrderStep2.TcPOU
// Struckig
// Copyright (C) 2022 Stefan Besler

// This program is free software: you can redistribute it and/or modify
// it under the terms of the GNU General Public License as published by
// the Free Software Foundation, either version 3 of the License, or
// (at your option) any later version.

// This program is distributed in the hope that it will be useful,
// but WITHOUT ANY WARRANTY; without even the implied warranty of
// MERCHANTABILITY or FITNESS FOR A PARTICULAR PURPOSE.  See the
// GNU General Public License for more details.
//
// You should have received a copy of the GNU General Public License
// along with THIS PROGRAM.  IF NOT, see <http://www.gnu.org/licenses/>.
/// Mathematical equations for Step 2 in third-order position interface: Time synchronization
FUNCTION_BLOCK INTERNAL PositionSecondOrderStep2
VAR
  minimize_jerk : BOOL;
  v0, a0 : LREAL;
  tf, vf, af : LREAL;
  _vMax, _vMin, _aMax, _aMin : LREAL;
  
  // Pre-calculated expressions
  pd : LREAL;
  tf_tf, tf_p3, tf_p4 : LREAL;
  vd, vd_vd : LREAL;
  ad, ad_ad : LREAL;
  v0_v0, vf_vf : LREAL;
  a0_a0, a0_p3, a0_p4, a0_p5, a0_p6 : LREAL;
  af_af, af_p3, af_p4, af_p5, af_p6 : LREAL;
  jMax_jMax : LREAL;
  g1, g2 : LREAL;
  t_min, t_max : LREAL;
  up_first : BOOL;
  
  d_extremasCount : INT;
  d_extremas : ARRAY[0..6] OF LREAL;
  indices : ARRAY[0..6] OF INT;
  
  h0, h0a, h0b, h0c, h1, h2 : LREAL;  
  h3, jf : LREAL;  
  ph1, ph2, ph3, ph4 : LREAL;
  t : LREAL; 
  orig, deriv : LREAL;
  i : INT;
  ph0, ph5, ph6, ph7 : LREAL;
  h1a : LREAL;
  p1, val_max : LREAL;
  polynom, deriva, dderiv, ddderiv, root : ARRAY[0..6] OF LREAL;
  dd_tz_intervals : ARRAY[0..6, 0..1] OF LREAL;
  tz, tz_max, tz_current, dd_tz_current, tz_min : LREAL; 
  deriv_newton, res, p_val, val_new : LREAL;    
END_VAR

METHOD CheckAll : BOOL
VAR_INPUT
  profile : REFERENCE TO ProfileDesc;
  vMax, vMin, aMax, aMin : LREAL;  
END_VAR
CheckAll := time_acc0(profile, vMax, vMin, aMax, aMin) OR_ELSE
            time_none(profile, vMax, vMin, aMax, aMin);
END_METHOD

METHOD Get : BOOL
VAR_INPUT
  Profile : REFERENCE TO ProfileDesc;
END_VAR
// Test all cases to get ones that match
// However we should guess which one is correct and try them first...
IF pd > 0
THEN
  Get := CheckAll(profile, _vMax, _vMin, _aMax, _aMin) OR_ELSE CheckAll(profile, _vMin, _vMax, _aMin, _aMax);
  RETURN;
END_IF

Get := CheckAll(profile, _vMin, _vMax, _aMin, _aMax) OR_ELSE CheckAll(profile, _vMax, _vMin, _aMax, _aMin);
END_METHOD

METHOD Set
VAR_INPUT
  tf : LREAL;
  p0, v0 : LREAL;
  pf, vf : LREAL;
  vMax, vMin : LREAL;
  aMax, aMin : LREAL;
END_VAR
THIS^.tf := tf;
THIS^.v0 := v0;
THIS^.vf := vf;
THIS^._vMax := vMax;
THIS^._vMin := vMin;
THIS^._aMax := aMax;
THIS^._aMin := aMin;

pd := pf - p0;
vd := vf - v0;
END_METHOD

METHOD PRIVATE time_acc0 : BOOL
VAR_INPUT
  profile : REFERENCE TO ProfileDesc;
  vMax, vMin, aMax, aMin : LREAL;
END_VAR
h1 := (2*aMax*(pd - tf*vf) - 2*aMin*(pd - tf*v0) + vd*vd)/(aMax*aMin) + tf*tf;
IF h1 >= 0
THEN
  h1 := SQRT(h1);

  profile.t[0] := (aMax*vd - aMax*aMin*(tf - h1))/(aMax*(aMax - aMin));
  profile.t[1] := h1;
  profile.t[2] := tf - (profile.t[0] + h1);
  profile.t[3] := 0;
  profile.t[4] := 0;
  profile.t[5] := 0;
  profile.t[6] := 0;

  IF profile.CheckForSecondOrderWithTiming(ProfileControlSigns.Uddu, ReachedLimits.Acc0, tf, aMax, aMin, vMax, vMin)
  THEN
    profile.pf := profile.p[7];
    time_acc0 := TRUE;
    RETURN;
  END_IF
END_IF


// UU Solution
h1 := (-vd + aMax*tf);
IF ABS(h1) > Constants.Epsilon AND_THEN ABS(2*aMax*h1) > Constants.Epsilon
THEN

  profile.t[0] := -vd*vd/(2*aMax*h1) + (pd - v0*tf)/h1;
  profile.t[1] := -vd/aMax + tf;
  profile.t[2] := 0;
  profile.t[3] := 0;
  profile.t[4] := 0;
  profile.t[5] := 0;
  profile.t[6] := tf - (profile.t[0] + profile.t[1]);
  
  IF profile.CheckForSecondOrderWithTiming(ProfileControlSigns.Uddu, ReachedLimits.Acc0, tf, aMax, aMin, vMax, vMin)
  THEN
    profile.pf := profile.p[7];
    time_acc0 := TRUE;
    RETURN;
  END_IF
END_IF


// UU Solution - 2 step
profile.t[0] := 0;
profile.t[1] := -vd/aMax + tf;
profile.t[2] := 0;
profile.t[3] := 0;
profile.t[4] := 0;
profile.t[5] := 0;
profile.t[6] := vd/aMax;

IF profile.CheckForSecondOrderWithTiming(ProfileControlSigns.Uddu, ReachedLimits.Acc0, tf, aMax, aMin, vMax, vMin)
THEN
  profile.pf := profile.p[7];
  time_acc0 := TRUE;
  RETURN;
END_IF
END_METHOD

/// Only for numerical issues, always return_after_found
METHOD PRIVATE time_none : BOOL
VAR_INPUT
  profile : REFERENCE TO ProfileDesc;
  vMax, vMin, aMax, aMin : LREAL;
END_VAR
IF ABS(v0) < Constants.DoubleEpsilon AND_THEN ABS(vf) < Constants.DoubleEpsilon AND_THEN ABS(pd) < Constants.DoubleEpsilon
THEN
  profile.t[0] := 0;
  profile.t[1] := tf;
  profile.t[2] := 0;
  profile.t[3] := 0;
  profile.t[4] := 0;
  profile.t[5] := 0;
  profile.t[6] := 0;

  IF profile.CheckForSecondOrderWithTiming(ProfileControlSigns.Uddu, ReachedLimits.None, tf, aMax, aMin, vMax, vMin)
  THEN
    profile.pf := profile.p[7];
    time_none := TRUE;
    RETURN;        
  END_IF
END_IF

// UD Solution 1/2
h1 := 2*(vf*tf - pd);

IF ABS(vd) > Constants.DoubleEpsilon AND_THEN ABS(h1) > Constants.Epsilon
THEN
  profile.t[0] := h1/vd;
  profile.t[1] := tf - profile.t[0];
  profile.t[2] := 0;
  profile.t[3] := 0;
  profile.t[4] := 0;
  profile.t[5] := 0;
  profile.t[6] := 0;

  af := vd*vd/h1;

  IF ((aMin - 1E-12 < af) AND_THEN (af < aMax + 1E-12) AND_THEN profile.CheckForSecondOrderWithTiming(ProfileControlSigns.Uddu, ReachedLimits.None, tf, af, -af, vMax, vMin))
  THEN
    profile.pf := profile.p[7];
    time_none := TRUE;
    RETURN;        
  END_IF
END_IF
END_METHOD

END_FUNCTION_BLOCK

// ---- Struckig/Velocity/VelocitySecondOrderStep1.TcPOU
// Struckig
// Copyright (C) 2022 Stefan Besler

// This program is free software: you can redistribute it and/or modify
// it under the terms of the GNU General Public License as published by
// the Free Software Foundation, either version 3 of the License, or
// (at your option) any later version.

// This program is distributed in the hope that it will be useful,
// but WITHOUT ANY WARRANTY; without even the implied warranty of
// MERCHANTABILITY or FITNESS FOR A PARTICULAR PURPOSE.  See the
// GNU General Public License for more details.
//
// You should have received a copy of the GNU General Public License
// along with THIS PROGRAM.  IF NOT, see <http://www.gnu.org/licenses/>.
/// Mathematical equations for Step 1 in second-order velocity interface: Extremal profiles
FUNCTION_BLOCK INTERNAL VelocitySecondOrderStep1 
VAR
  _aMax : LREAL;
  _aMin : LREAL;
  vd : LREAL;
END_VAR

METHOD Get : BOOL
VAR_INPUT
  input : ProfileDesc;
END_VAR
VAR_IN_OUT
  block : Block; 
END_VAR
VAR
  p : REFERENCE TO ProfileDesc;
  af : LREAL;
END_VAR
p REF= block.Pmin;
p.SetBoundary(input);

af := SEL(vd > 0, _aMin, _aMax);
p.t[0] := 0;
p.t[1] := vd / af;
p.t[2] := 0;
p.t[3] := 0;
p.t[4] := 0;
p.t[5] := 0;
p.t[6] := 0;

IF p.CheckForSecondOrderVelocity(ProfileControlSigns.Uddu, ReachedLimits.Acc0, af)
THEN
  block.Tmin := p.t_sum[6] + p.Brake.Duration + p.Accel.Duration;
  Get := TRUE;
  RETURN;
END_IF
END_METHOD

METHOD Set
VAR_INPUT
  v0, vf : LREAL; 
  aMax, aMin : LREAL;  
END_VAR
THIS^._aMax := aMax;
THIS^._aMin := aMin;
THIS^.vd := vf - v0;
END_METHOD

END_FUNCTION_BLOCK

// ---- Struckig/Velocity/VelocitySecondOrderStep2.TcPOU
// Struckig
// Copyright (C) 2022 Stefan Besler

// This program is free software: you can redistribute it and/or modify
// it under the terms of the GNU General Public License as published by
// the Free Software Foundation, either version 3 of the License, or
// (at your option) any later version.

// This program is distributed in the hope that it will be useful,
// but WITHOUT ANY WARRANTY; without even the implied warranty of
// MERCHANTABILITY or FITNESS FOR A PARTICULAR PURPOSE.  See the
// GNU General Public License for more details.
//
// You should have received a copy of the GNU General Public License
// along with THIS PROGRAM.  IF NOT, see <http://www.gnu.org/licenses/>.
/// Mathematical equations for Step 2 in second-order velocity interface: Time synchronization
FUNCTION_BLOCK INTERNAL VelocitySecondOrderStep2 
VAR
  _aMax : LREAL;
  _aMin : LREAL;
  tf : LREAL;
  vd : LREAL;
END_VAR

METHOD Get : BOOL
VAR_INPUT
  profile : ProfileDesc;
END_VAR
VAR
  af : LREAL;
END_VAR
af := vd / tf;
profile.t[0] := 0;
profile.t[1] := tf;
profile.t[2] := 0;
profile.t[3] := 0;
profile.t[4] := 0;
profile.t[5] := 0;
profile.t[6] := 0;

IF profile.CheckForSecondOrderVelocityWithTiming2(ProfileControlSigns.Uddu, ReachedLimits.None, tf, af, _aMax, _aMin)
THEN
  profile.pf := profile.p[6];
  Get := TRUE;
  RETURN;
END_IF
END_METHOD

METHOD Set
VAR_INPUT
  tf : LREAL;
  v0, vf : LREAL; 
  aMax, aMin : LREAL;  
END_VAR
THIS^._aMax := aMax;
THIS^._aMin := aMin;
THIS^.tf := tf;
THIS^.vd := vf - v0;
END_METHOD

END_FUNCTION_BLOCK

// ---- Struckig/Position/PositionFirstOrderStep1.TcPOU
// Struckig
// Copyright (C) 2022 Stefan Besler

// This program is free software: you can redistribute it and/or modify
// it under the terms of the GNU General Public License as published by
// the Free Software Foundation, either version 3 of the License, or
// (at your option) any later version.

// This program is distributed in the hope that it will be useful,
// but WITHOUT ANY WARRANTY; without even the implied warranty of
// MERCHANTABILITY or FITNESS FOR A PARTICULAR PURPOSE.  See the
// GNU General Public License for more details.
//
// You should have received a copy of the GNU General Public License
// along with THIS PROGRAM.  IF NOT, see <http://www.gnu.org/licenses/>.
/// Mathematical equations for Step 1 in third-order position interface: Extremal profiles
FUNCTION_BLOCK INTERNAL PositionFirstOrderStep1
VAR
  v0 : LREAL;
  vf : LREAL;
  _vMax, _vMin : LREAL;

  // Pre-calculated expressions
  pd : LREAL;  
END_VAR

METHOD Get : BOOL
VAR_INPUT
  input : REFERENCE TO ProfileDesc;
  block : REFERENCE TO Block; 
END_VAR
VAR_INST
  vMax, vMin, aMax, aMin, jMax : LREAL;
  profile : REFERENCE TO ProfileDesc;
END_VAR
profile REF= block.Pmin;
profile.SetBoundary(input);

vf := SEL(pd > 0, _vMin, _vMax);
profile.t[0] := 0;
profile.t[1] := 0;
profile.t[2] := 0;
profile.t[3] := pd / vf;
profile.t[4] := 0;
profile.t[5] := 0;
profile.t[6] := 0;

IF profile.CheckForFirstOrder(ProfileControlSigns.Uddu, ReachedLimits.Vel, vf)
THEN
  block.Tmin := block.Pmin.t_sum[6] + block.Pmin.Brake.Duration + block.Pmin.Accel.Duration;
  Get := TRUE;
END_IF
END_METHOD

METHOD Set
VAR_INPUT
  p0 : LREAL;
  pf : LREAL;
  vMax, vMin : LREAL;
END_VAR
THIS^.v0 := v0;
THIS^.vf := vf;
THIS^._vMax := vMax;
THIS^._vMin := vMin;

pd := pf - p0;
END_METHOD

END_FUNCTION_BLOCK

// ---- Struckig/Position/PositionFirstOrderStep2.TcPOU
// Struckig
// Copyright (C) 2022 Stefan Besler

// This program is free software: you can redistribute it and/or modify
// it under the terms of the GNU General Public License as published by
// the Free Software Foundation, either version 3 of the License, or
// (at your option) any later version.

// This program is distributed in the hope that it will be useful,
// but WITHOUT ANY WARRANTY; without even the implied warranty of
// MERCHANTABILITY or FITNESS FOR A PARTICULAR PURPOSE.  See the
// GNU General Public License for more details.
//
// You should have received a copy of the GNU General Public License
// along with THIS PROGRAM.  IF NOT, see <http://www.gnu.org/licenses/>.
/// Mathematical equations for Step 2 in third-order position interface: Time synchronization
FUNCTION_BLOCK INTERNAL PositionFirstOrderStep2
VAR
  minimize_jerk : BOOL;
  v0, a0 : LREAL;
  tf, vf, af : LREAL;
  _vMax, _vMin : LREAL;
  
  // Pre-calculated expressions
  pd : LREAL;
  tf_tf, tf_p3, tf_p4 : LREAL;
  vd, vd_vd : LREAL;
  ad, ad_ad : LREAL;
  v0_v0, vf_vf : LREAL;
  a0_a0, a0_p3, a0_p4, a0_p5, a0_p6 : LREAL;
  af_af, af_p3, af_p4, af_p5, af_p6 : LREAL;
  jMax_jMax : LREAL;
  g1, g2 : LREAL;
  t_min, t_max : LREAL;
  up_first : BOOL;
  
  d_extremasCount : INT;
  d_extremas : ARRAY[0..6] OF LREAL;
  indices : ARRAY[0..6] OF INT;
  
  h0, h0a, h0b, h0c, h1, h2 : LREAL;  
  h3, jf : LREAL;  
  ph1, ph2, ph3, ph4 : LREAL;
  t : LREAL; 
  orig, deriv : LREAL;
  i : INT;
  ph0, ph5, ph6, ph7 : LREAL;
  h1a : LREAL;
  p1, val_max : LREAL;
  polynom, deriva, dderiv, ddderiv, root : ARRAY[0..6] OF LREAL;
  dd_tz_intervals : ARRAY[0..6, 0..1] OF LREAL;
  tz, tz_max, tz_current, dd_tz_current, tz_min : LREAL; 
  deriv_newton, res, p_val, val_new : LREAL;    
END_VAR

METHOD Get : BOOL
VAR_INPUT
  profile : REFERENCE TO ProfileDesc;
END_VAR
vf := pd / tf;

profile.t[0] := 0;
profile.t[1] := 0;
profile.t[2] := 0;
profile.t[3] := tf;
profile.t[4] := 0;
profile.t[5] := 0;
profile.t[6] := 0;

Get := profile.CheckForFirstOrderWithTiming2(ProfileControlSigns.Uddu, ReachedLimits.None, tf, vf, _vMax, _vMin);
END_METHOD

METHOD Set
VAR_INPUT
  tf : LREAL;
  p0 : LREAL;
  pf : LREAL;
  vMax, vMin : LREAL;
END_VAR
THIS^.tf := tf;
THIS^.v0 := v0;
THIS^.vf := vf;
THIS^._vMax := vMax;
THIS^._vMin := vMin;

pd := pf - p0;
vd := vf - v0;
END_METHOD

END_FUNCTION_BLOCK

// ---- Struckig/Math/IsInfinity.TcPOU
// Struckig
// Copyright (C) 2022 Stefan Besler

// This program is free software: you can redistribute it and/or modify
// it under the terms of the GNU General Public License as published by
// the Free Software Foundation, either version 3 of the License, or
// (at your option) any later version.

// This program is distributed in the hope that it will be useful,
// but WITHOUT ANY WARRANTY; without even the implied warranty of
// MERCHANTABILITY or FITNESS FOR A PARTICULAR PURPOSE.  See the
// GNU General Public License for more details.
//
// You should have received a copy of the GNU General Public License
// along with THIS PROGRAM.  IF NOT, see <http://www.gnu.org/licenses/>.
/// Checks whether a floating-point value is positive or negative infinity.
FUNCTION IsInfinity : BOOL
VAR_INPUT
  value : LREAL; //< Input value.
END_VAR

IsInfinity := value = Constants.Infinity OR_ELSE value = -Constants.Infinity;

END_FUNCTION

// ---- Struckig/Math/Fmod.TcPOU
// Struckig
// Copyright (C) 2022 Stefan Besler

// This program is free software: you can redistribute it and/or modify
// it under the terms of the GNU General Public License as published by
// the Free Software Foundation, either version 3 of the License, or
// (at your option) any later version.

// This program is distributed in the hope that it will be useful,
// but WITHOUT ANY WARRANTY; without even the implied warranty of
// MERCHANTABILITY or FITNESS FOR A PARTICULAR PURPOSE.  See the
// GNU General Public License for more details.
//
// You should have received a copy of the GNU General Public License
// along with THIS PROGRAM.  IF NOT, see <http://www.gnu.org/licenses/>.
/// Floating-point remainder operation.
/// Returns the remainder of `x / y` with truncation toward zero:
/// `x - TRUNC(x / y) * y`.
FUNCTION Fmod : LREAL
VAR_INPUT
  x : LREAL; //< Dividend.
  y : LREAL; //< Divisor.
END_VAR

Fmod := x - TRUNC(x / y) * y;

END_FUNCTION

// ---- Struckig/Otg1.TcPOU
// Struckig
// Copyright (C) 2022 Stefan Besler

// This program is free software: you can redistribute it and/or modify
// it under the terms of the GNU General Public License as published by
// the Free Software Foundation, either version 3 of the License, or
// (at your option) any later version.

// This program is distributed in the hope that it will be useful,
// but WITHOUT ANY WARRANTY; without even the implied warranty of
// MERCHANTABILITY or FITNESS FOR A PARTICULAR PURPOSE.  See the
// GNU General Public License for more details.
//
// You should have received a copy of the GNU General Public License
// along with THIS PROGRAM.  IF NOT, see <http://www.gnu.org/licenses/>.
{attribute 'conditionalshow_all_locals'}
/// Convenience wrapper for single-DoF trajectory generation.
/// This function block forwards all calls to an internal `Otg` instance with `Dofs = 1`.
/// Use this block when your application controls exactly one axis and you want
/// scalar I/O instead of vectors.
///
/// ```st
/// otg1(
///   CycleTime := 0.001,
///   ControlInterface := ControlInterfaceType.Position,
///   Synchronization := SynchronizationType.TimeSync
/// );
/// Axis.Setpoint := otg1.NewPosition;
/// ```
FUNCTION_BLOCK Otg1 IMPLEMENTS IOtg
VAR_INPUT
  CycleTime : LREAL;
  ControlInterface : ControlInterfaceType := ControlInterfaceType.Position; //< The default position interface controls the full kinematic state.
  Synchronization : SynchronizationType := SynchronizationType.TimeSync; //< Synchronization behavior of multiple DoFs
  PerDofControlInterface : ControlInterfaceType; //< Per-DoF control interface (overwrites global ControlInterface)
  PerDofSynchronization :  SynchronizationType; //< Per-DoF synchronization (overwrites global Synchronization)
  Discretization : DiscretizationType; //< Whether the duration should be a discrete multiple of the control cycle (off by default)
  CurrentPosition, CurrentVelocity, CurrentAcceleration : LREAL; //< Current state
  TargetPosition, TargetVelocity, TargetAcceleration : LREAL; //< Target state
  MaxVelocity, MaxAcceleration, MaxJerk : LREAL; //< Kinematic constraints
  MinVelocity, MinAcceleration : LREAL; //< Optional kindematic constraints
  MinDuration : LREAL := 0; //< Optional minimum duration of a trajectory. This is only considered if the Synchronization type is not none
  EnableAutoPropagate : BOOL; //< If set to true, PassOutputToInput is automatically called internally after calling the function block's body
  SmoothBrake : BOOL := ParameterList.SmoothBrake; //< See Otg.SmoothBrake
END_VAR
VAR_OUTPUT
  NewPosition, NewVelocity, NewAcceleration, NewJerk : LREAL;
  NewCalculation : BOOL; //< Was a new trajectory calculation performed in the last cycle?
  CurrentTime : LREAL; //< Time elapsed on the current trajectory in seconds.
END_VAR
VAR
  _otg : Otg(0,0);
END_VAR

_otg.PerDofControlInterface[0] := PerDofControlInterface;
_otg.PerDofSynchronization[0] := PerDofSynchronization;
_otg.Discretization := Discretization;
_otg.CurrentPosition[0] := CurrentPosition;
_otg.CurrentVelocity[0] := CurrentVelocity;
_otg.CurrentAcceleration[0] := CurrentAcceleration;
_otg.TargetPosition[0] := TargetPosition;
_otg.TargetVelocity[0] := TargetVelocity;
_otg.TargetAcceleration[0] := TargetAcceleration;
_otg.MaxVelocity[0] := MaxVelocity;
_otg.MaxAcceleration[0] := MaxAcceleration;
_otg.MaxJerk[0] := MaxJerk;
_otg.MinVelocity[0] := MinVelocity;
_otg.MinAcceleration[0] := MinAcceleration;
_otg.MinDuration := MinDuration;
_otg.EnableAutoPropagate := EnableAutoPropagate;
_otg.SmoothBrake := SmoothBrake;

_otg(CycleTime := CycleTime,
     Dofs := 1,
     ControlInterface := ControlInterface,
     Synchronization := Synchronization);
     
CurrentPosition := _otg.CurrentPosition[0];
CurrentVelocity := _otg.CurrentVelocity[0];
CurrentAcceleration := _otg.CurrentAcceleration[0];     
NewPosition := _otg.NewPosition[0];
NewVelocity := _otg.NewVelocity[0];
NewAcceleration := _otg.NewAcceleration[0];
NewJerk := _otg.NewJerk[0];
CurrentTime := _otg.CurrentTime;

/// \copydoc Struckig.Otg#AtTime
{attribute 'conditionalshow'}
METHOD AtTime
VAR_INPUT
  t : LREAL;
  new_position : POINTER TO LREAL;
  new_velocity : POINTER TO LREAL;
  new_acceleration : POINTER TO LREAL;
  new_jerk : POINTER TO LREAL;
  new_section : POINTER TO INT;
END_VAR
_otg.AtTime(t, new_position, new_velocity, new_acceleration, new_jerk, new_section);
END_METHOD

/// \copydoc Struckig.Otg#AtTime1
{attribute 'conditionalshow'}
METHOD AtTime1
VAR_INPUT
  t : LREAL;
  new_position : REFERENCE TO LREAL;
  new_velocity : REFERENCE TO LREAL;
  new_acceleration : REFERENCE TO LREAL;
  new_jerk : REFERENCE TO LREAL;  
END_VAR
_otg.AtTime1(t, new_position, new_velocity, new_acceleration, new_jerk);
END_METHOD

/// \copydoc Struckig.Otg#Cyclic
METHOD Cyclic
VAR_INPUT
END_VAR
_otg();
END_METHOD

/// \copydoc Struckig.Otg#Duration
PROPERTY Duration : LREAL
GET
Duration := _otg.Duration;
END_GET
END_PROPERTY

/// \copydoc Struckig.Otg#ErrorCode
METHOD ErrorCode : TrajectoryErrorCode
VAR_INPUT
END_VAR
ErrorCode := _otg.ErrorCode();
END_METHOD

/// \copydoc Struckig.Otg#ErrorMessage
METHOD ErrorMessage : STRING(255)
VAR_INPUT
END_VAR
ErrorMessage := _otg.ErrorMessage();
END_METHOD

METHOD FB_init : BOOL
VAR_INPUT
	bInitRetains : BOOL; // if TRUE, the retain variables are initialized (warm start / cold start)
	bInCopyCode : BOOL;  // if TRUE, the instance afterwards gets moved into the copy code (online change)
  cycletime : LREAL;
END_VAR
_otg.FB_init(bInitRetains, bInCopyCode, cycletime, 1);
THIS^.CycleTime := cycletime;
END_METHOD

/// \copydoc Struckig.Otg#PassOutputToInput
METHOD PassOutputToInput
VAR_INPUT
END_VAR
_otg.PassOutputToInput();
END_METHOD

/// \copydoc Struckig.Otg#Reset
METHOD Reset
VAR_INPUT
END_VAR
_otg.Reset();
END_METHOD

/// \copydoc Struckig.Otg#State
PROPERTY State : TrajectoryState
GET
State := _otg.State;
END_GET
END_PROPERTY

/// \copydoc Struckig.Otg#ValidateInput
{attribute 'conditionalshow'}
METHOD ValidateInput : BOOL
VAR_INPUT
  checkCurrentStateWithinLimits : BOOL;
  checkTargetStateWithinLimits : BOOL;
END_VAR
_otg.ValidateInput(checkCurrentStateWithinLimits, checkTargetStateWithinLimits);
END_METHOD

END_FUNCTION_BLOCK

// ---- Struckig/Math/Ceil.TcPOU
// Struckig
// Copyright (C) 2022 Stefan Besler

// This program is free software: you can redistribute it and/or modify
// it under the terms of the GNU General Public License as published by
// the Free Software Foundation, either version 3 of the License, or
// (at your option) any later version.

// This program is distributed in the hope that it will be useful,
// but WITHOUT ANY WARRANTY; without even the implied warranty of
// MERCHANTABILITY or FITNESS FOR A PARTICULAR PURPOSE.  See the
// GNU General Public License for more details.
//
// You should have received a copy of the GNU General Public License
// along with THIS PROGRAM.  IF NOT, see <http://www.gnu.org/licenses/>.
/// Returns the smallest integer value greater than or equal to `val`.
/// NaN and +/-Infinity are passed through unchanged.
FUNCTION Ceil : LREAL
VAR_INPUT
  val : LREAL; //< Input value.
END_VAR
VAR CONSTANT
  InfinityBits : ULINT := ULINT#16#7FF0000000000000;
END_VAR
VAR
  InfinityPtr : POINTER TO LREAL := ADR(InfinityBits);
END_VAR

IF val <> val OR_ELSE val = InfinityPtr^ OR_ELSE val = -InfinityPtr^ // nan or inf
THEN
  RETURN;
END_IF

Ceil := DINT_TO_LREAL(LREAL_TO_DINT(val));
IF Ceil < val THEN
	Ceil := Ceil + 1;
END_IF;

END_FUNCTION

// ---- Struckig/Math/IsNaN.TcPOU
// Struckig
// Copyright (C) 2022 Stefan Besler

// This program is free software: you can redistribute it and/or modify
// it under the terms of the GNU General Public License as published by
// the Free Software Foundation, either version 3 of the License, or
// (at your option) any later version.

// This program is distributed in the hope that it will be useful,
// but WITHOUT ANY WARRANTY; without even the implied warranty of
// MERCHANTABILITY or FITNESS FOR A PARTICULAR PURPOSE.  See the
// GNU General Public License for more details.
//
// You should have received a copy of the GNU General Public License
// along with THIS PROGRAM.  IF NOT, see <http://www.gnu.org/licenses/>.
/// Checks whether a floating-point value is NaN.
/// Uses the IEEE-754 property that NaN is not equal to itself.
FUNCTION IsNaN : BOOL
VAR_INPUT
  value : LREAL; //< Input value.
END_VAR

IsNaN := value <> value;

END_FUNCTION

// ---- Struckig/Math/Power.TcPOU
// Struckig
// Copyright (C) 2022 Stefan Besler

// This program is free software: you can redistribute it and/or modify
// it under the terms of the GNU General Public License as published by
// the Free Software Foundation, either version 3 of the License, or
// (at your option) any later version.

// This program is distributed in the hope that it will be useful,
// but WITHOUT ANY WARRANTY; without even the implied warranty of
// MERCHANTABILITY or FITNESS FOR A PARTICULAR PURPOSE.  See the
// GNU General Public License for more details.
//
// You should have received a copy of the GNU General Public License
// along with THIS PROGRAM.  IF NOT, see <http://www.gnu.org/licenses/>.
/// Internal power helper that preserves sign for negative bases.
/// Evaluates `sign(v) * |v|^e`.
FUNCTION INTERNAL Power : LREAL
VAR_INPUT
  v : LREAL; //< Base value.
  e : LREAL; //< Exponent.
END_VAR

Power := SEL(v < 0, 1.0, -1.0) * EXPT(ABS(v), e);

END_FUNCTION
